{attribute 'qualified_only'}
{attribute 'strict'}
TYPE EStampStates :
(
	none := 0,
	unpressed := 1,
	pressed := 2
) UINT;
END_TYPE

(* stored: Version 1.1.0.1, ProductVersion 3.1.4024.9
   DUT EStampStates: Id {34643114-d342-40d9-9926-dc7af836af2b} *)
